(* Logix 5000 project; controller CarbonScout_MK6 vendor 1 type 14 code 154 rev 32.11; software revision 32.00; part 13 of 17 *)
(* tags used below, declared in another part *)
   Data_TLSaver : BOOL;
   DN_Cal : BOOL;   // Calculation Done Bit to proceed next step
   Index : DINT;
   LocalSampleTank : DINT;
   ONS : BOOL[32];
   TimeCompare : TimerCompare;
   AI_LIT_01 : P_AIn;   // Carbon Scout Laser Level Transmitter
   AI_LIT_02 : P_AIn;   // Carbon Scout Cone Level Transmitter
   CS_CarbonSP : REAL;
   CS_DINTParams : DINT[100];
   CS_REALParams : REAL[80];   // CS REAL Parameters
   CS_Result : CS_Results;   // Sample Result Live Async
   CS_Results : CS_Results[20];   // Results Just for DataStore
   CS_ResultStore : CS_Results[20,20];   // Sample Result Historical
   CS_Seq : GEK_Sequence;
   CS_Seq_ControlStop : BOOL;
   CS_Tank : CS_TankParams[20];
   CS_Timer : TIMER[80];
   Data_constant1 : BOOL;
   Data_Saved : BOOL;
   Data_Saver : BOOL;
   Data_Trigger : BOOL;
   Data_Triggered : BOOL;
   Delete2_Trigger : BOOL;
   Delete_Trigger : BOOL;
   Email_Trigger : BOOL;
   Email_Trigger2 : BOOL;
   LeakCheck : BOOL;
   N51 : DINT[5];   // From Client
   Oneshot : DINT;
   Oneshot2 : DINT;
   Oneshot3 : DINT;
   Simulation : DINT;
   TankNum : DINT;
   TankPointer : DINT;
   TimeAndDate : DINT[7];
   Valve_XV_19 : P_ValveSO;   // Laser window
(* SeqProgram, continued *)

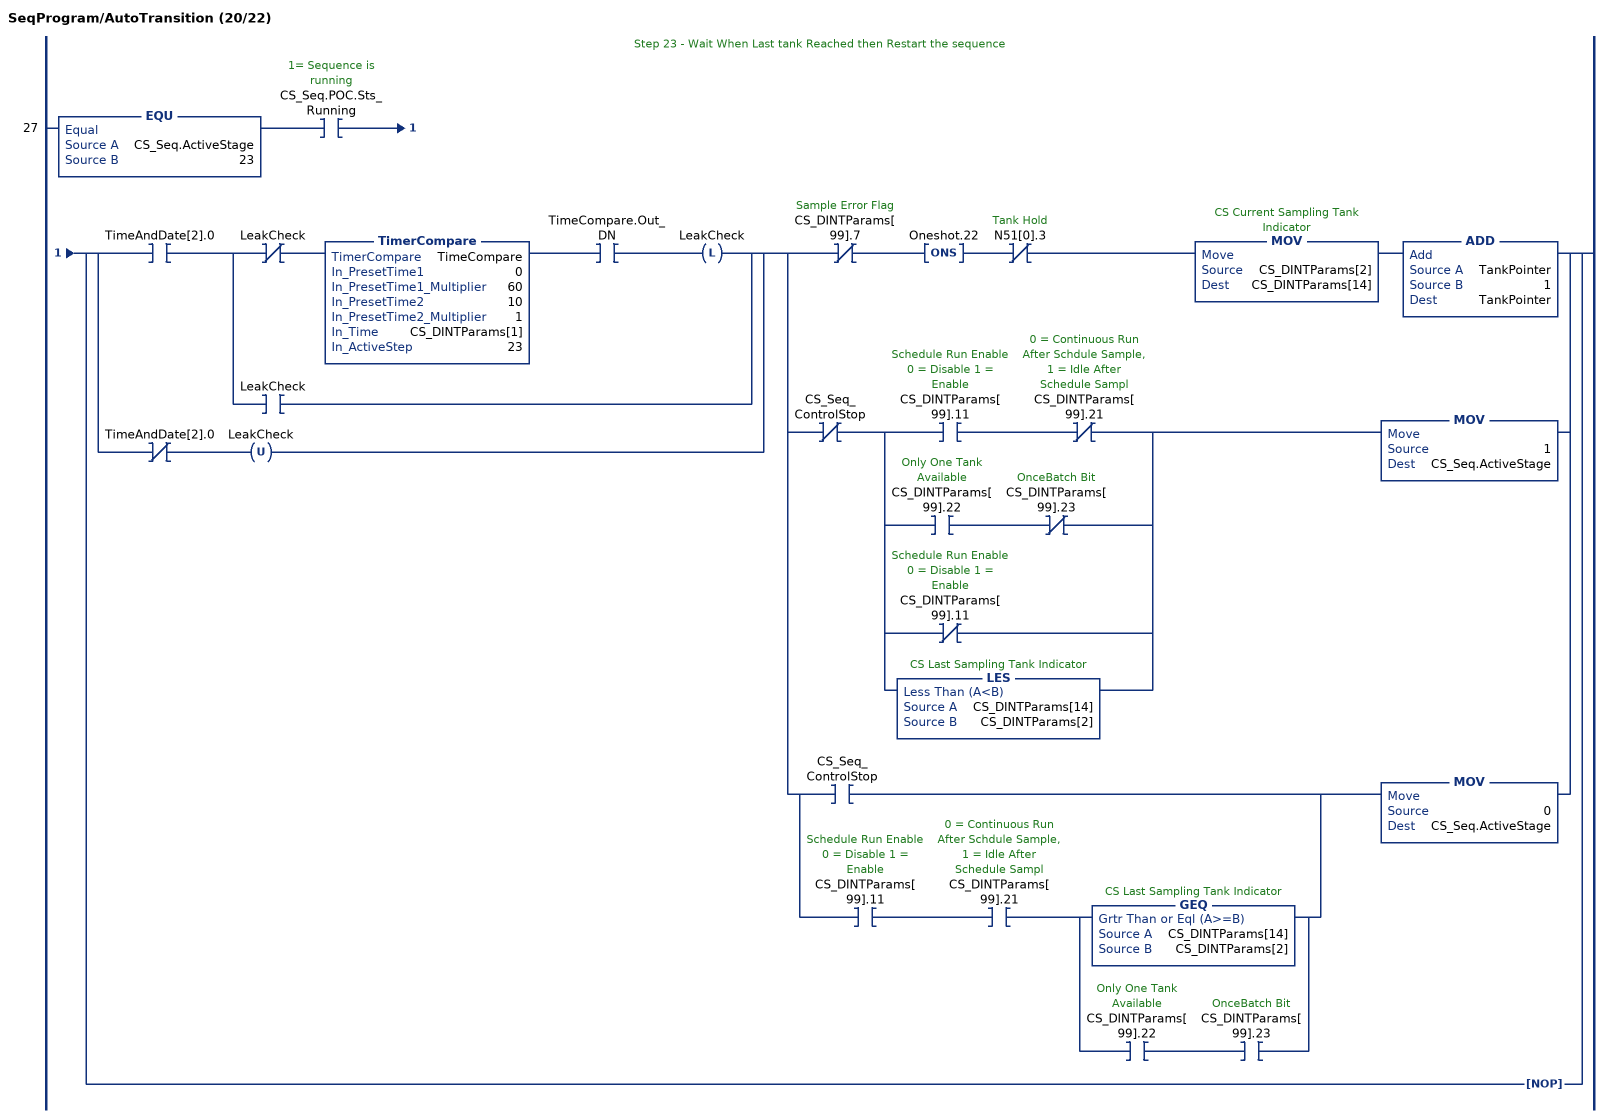
   [picture p263: SeqProgram/AutoTransition rungs 27-27]
   // Step 23 - Wait When Last tank Reached then Restart the sequence
   27: EQU(CS_Seq.ActiveStage,23)XIC(CS_Seq.POC.Sts_Running)[[XIC(TimeAndDate[2].0) [XIO(LeakCheck) TimerCompare(TimeCompare,0,60,10,1,CS_DINTParams[1],23) XIC(TimeCompare.Out_DN) OTL(LeakCheck) ,XIC(LeakCheck) ] ,XIO(TimeAndDate[2].0) OTU(LeakCheck) ] [XIO(CS_DINTParams[99].7) ONS(Oneshot.22) XIO(N51[0].3) MOV(CS_DINTParams[2],CS_DINTParams[14]) ADD(TankPointer,1,TankPointer) ,[XIO(CS_Seq_ControlStop) [XIC(CS_DINTParams[99].11) XIO(CS_DINTParams[99].21) ,[XIC(CS_DINTParams[99].22) XIO(CS_DINTParams[99].23) ,XIO(CS_DINTParams[99].11) ,LES(CS_DINTParams[14],CS_DINTParams[2]) ] ] MOV(1,CS_Seq.ActiveStage) ,[XIC(CS_Seq_ControlStop) ,XIC(CS_DINTParams[99].11) XIC(CS_DINTParams[99].21) [GEQ(CS_DINTParams[14],CS_DINTParams[2]) ,XIC(CS_DINTParams[99].22) XIC(CS_DINTParams[99].23) ] ] MOV(0,CS_Seq.ActiveStage) ] ] ,NOP() ];
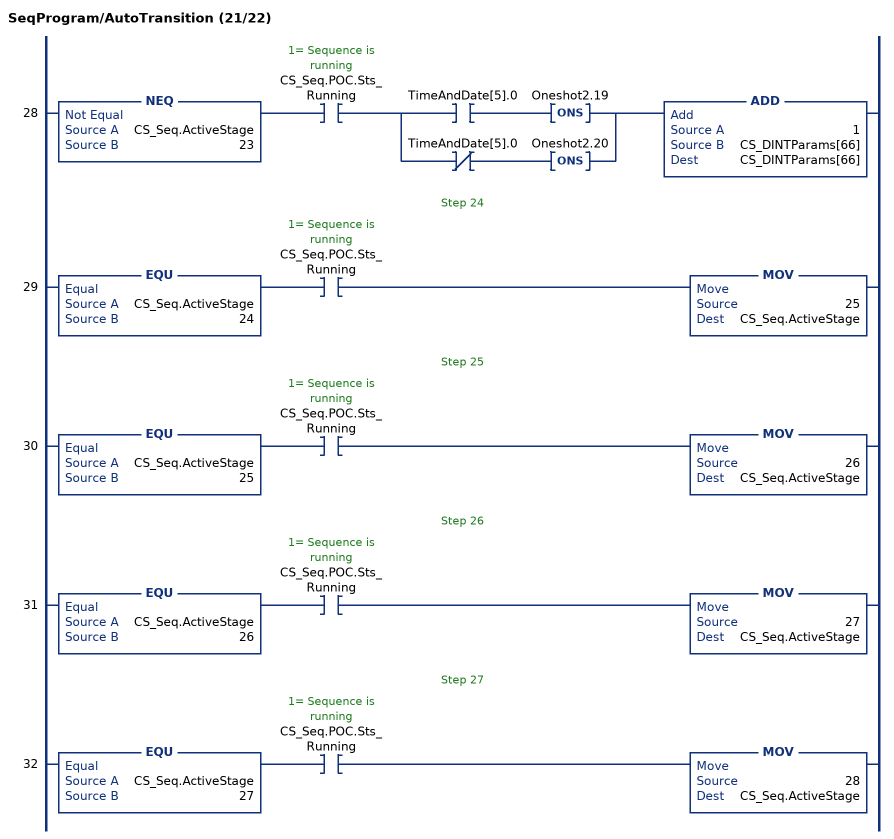
   28: NEQ(CS_Seq.ActiveStage,23)XIC(CS_Seq.POC.Sts_Running)[XIC(TimeAndDate[5].0) ONS(Oneshot2.19) ,XIO(TimeAndDate[5].0) ONS(Oneshot2.20) ]ADD(1,CS_DINTParams[66],CS_DINTParams[66]);
   // Step 24
   29: EQU(CS_Seq.ActiveStage,24)XIC(CS_Seq.POC.Sts_Running)MOV(25,CS_Seq.ActiveStage);
   // Step 25
   30: EQU(CS_Seq.ActiveStage,25)XIC(CS_Seq.POC.Sts_Running)MOV(26,CS_Seq.ActiveStage);
   // Step 26
   31: EQU(CS_Seq.ActiveStage,26)XIC(CS_Seq.POC.Sts_Running)MOV(27,CS_Seq.ActiveStage);
   // Step 27
   32: EQU(CS_Seq.ActiveStage,27)XIC(CS_Seq.POC.Sts_Running)MOV(28,CS_Seq.ActiveStage);
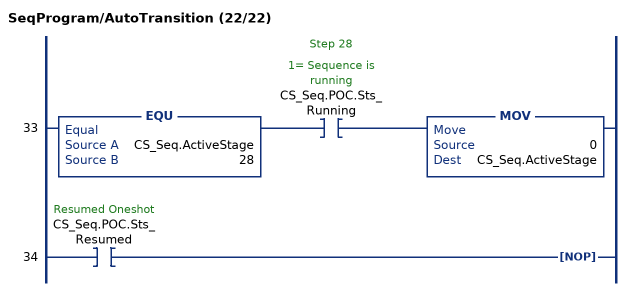
   // Step 28
   33: EQU(CS_Seq.ActiveStage,28)XIC(CS_Seq.POC.Sts_Running)MOV(0,CS_Seq.ActiveStage);
   34: XIC(CS_Seq.POC.Sts_Resumed)NOP();
END_ROUTINE

ROUTINE CarbonCals   (* ladder *)
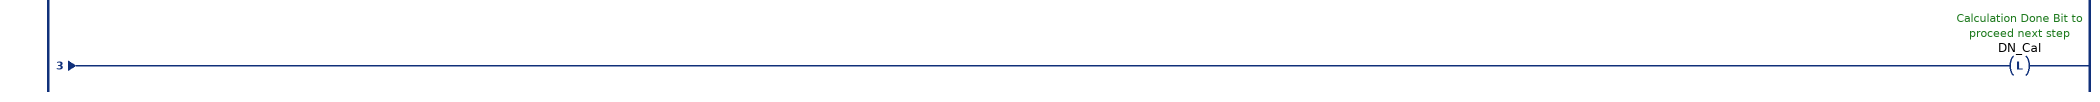
   // Calculating carbon volume
   0: EQU(CS_Seq.ActiveStage,14)XIO(CS_Tank[LocalSampleTank].LeachOnly)XIC(CS_Seq.POC.Sts_Running)[XIC(TimeCompare.Out_DN) [XIO(CS_DINTParams[93].20) [XIC(CS_DINTParams[93].8) ,XIC(CS_DINTParams[93].9) ] ,XIO(CS_DINTParams[99].15) ] ,XIC(CS_Timer[71].EN) ]TON(CS_Timer[71],?,?)XIC(CS_Timer[71].DN)ONS(Oneshot.23)[CPT(CS_REALParams[15],CS_REALParams[0]-CS_REALParams[1]) [CMP(CS_REALParams[15]<=0) CLR(CS_Result.Carbon_VOL_ml) ,CMP(CS_REALParams[15]>0) [CMP(CS_REALParams[15]<=CS_REALParams[14]) CPT(CS_Result.Carbon_VOL_ml,CS_REALParams[15]*(CS_REALParams[5]*CS_REALParams[5]/4)*3.1415927/1000) ,CMP(CS_REALParams[15]>CS_REALParams[14]) [CPT(CS_REALParams[17],CS_REALParams[14]*(CS_REALParams[5]*CS_REALParams[5]/4)*3.1415927) ,CPT(CS_REALParams[19],CS_REALParams[13]-CS_REALParams[14]) ,CPT(CS_REALParams[21],CS_REALParams[19]/(CS_REALParams[12]-CS_REALParams[5])) ,CPT(CS_REALParams[16],CS_REALParams[5]*CS_REALParams[21]) ,CPT(CS_REALParams[20],CS_REALParams[16]+(CS_REALParams[15]-CS_REALParams[14])) ,CPT(CS_REALParams[18],CS_REALParams[20]/CS_REALParams[21]) ] CPT(CS_Result.Carbon_VOL_ml,(CS_REALParams[17]+((CS_REALParams[18]*CS_REALParams[18]*3.1415927/4*CS_REALParams[20]-(CS_REALParams[5]*CS_REALParams[5]*3.1415927/4*CS_REALParams[16]))/3))/1000) ] ] ,DIV(CS_Result.Carbon_VOL_ml,CS_REALParams[11],CS_REALParams[51]) MOV(CS_REALParams[51],CS_Result.Carbon_mLperL) MUL(CS_Result.Carbon_VOL_ml,CS_REALParams[6],CS_Result.Carbon_MASS) ,MOV(LocalSampleTank,CS_Result.Sample_Tank) MOV(CS_REALParams[15],CS_Result.Carbon_Height) DIV(CS_Result.Carbon_MASS,CS_REALParams[11],CS_Result.Carbon_DIST) CPT(CS_Tank[LocalSampleTank].TotalCarbonMass,CS_Result.Carbon_DIST*CS_Tank[LocalSampleTank].Volume) CPT(CS_Tank[LocalSampleTank].GoldMass,CS_Tank[LocalSampleTank].TotalCarbonMass*CS_Result.Au) CPT(CS_Result.DisplacedCarbonVol,CS_REALParams[51]*(CS_Result.Sample_FlowRate*CS_Tank[LocalSampleTank].Sample_Time*0.4)) CPT(CS_Result.DisplacedCarbonMass,CS_Result.Sample_FlowRate*CS_Tank[LocalSampleTank].Sample_Time*0.4*CS_Result.Carbon_DIST) ,MOV(TimeAndDate[0],CS_Result.Year) MOV(TimeAndDate[1],CS_Result.Month) MOV(TimeAndDate[2],CS_Result.Day) MOV(TimeAndDate[3],CS_Result.Hour) MOV(TimeAndDate[4],CS_Result.Min) ,MOV(0,Index) FOR(DataShift,Index,0,18,1) CPS(CS_Result,CS_ResultStore[LocalSampleTank,0],1) ]OTL(DN_Cal);
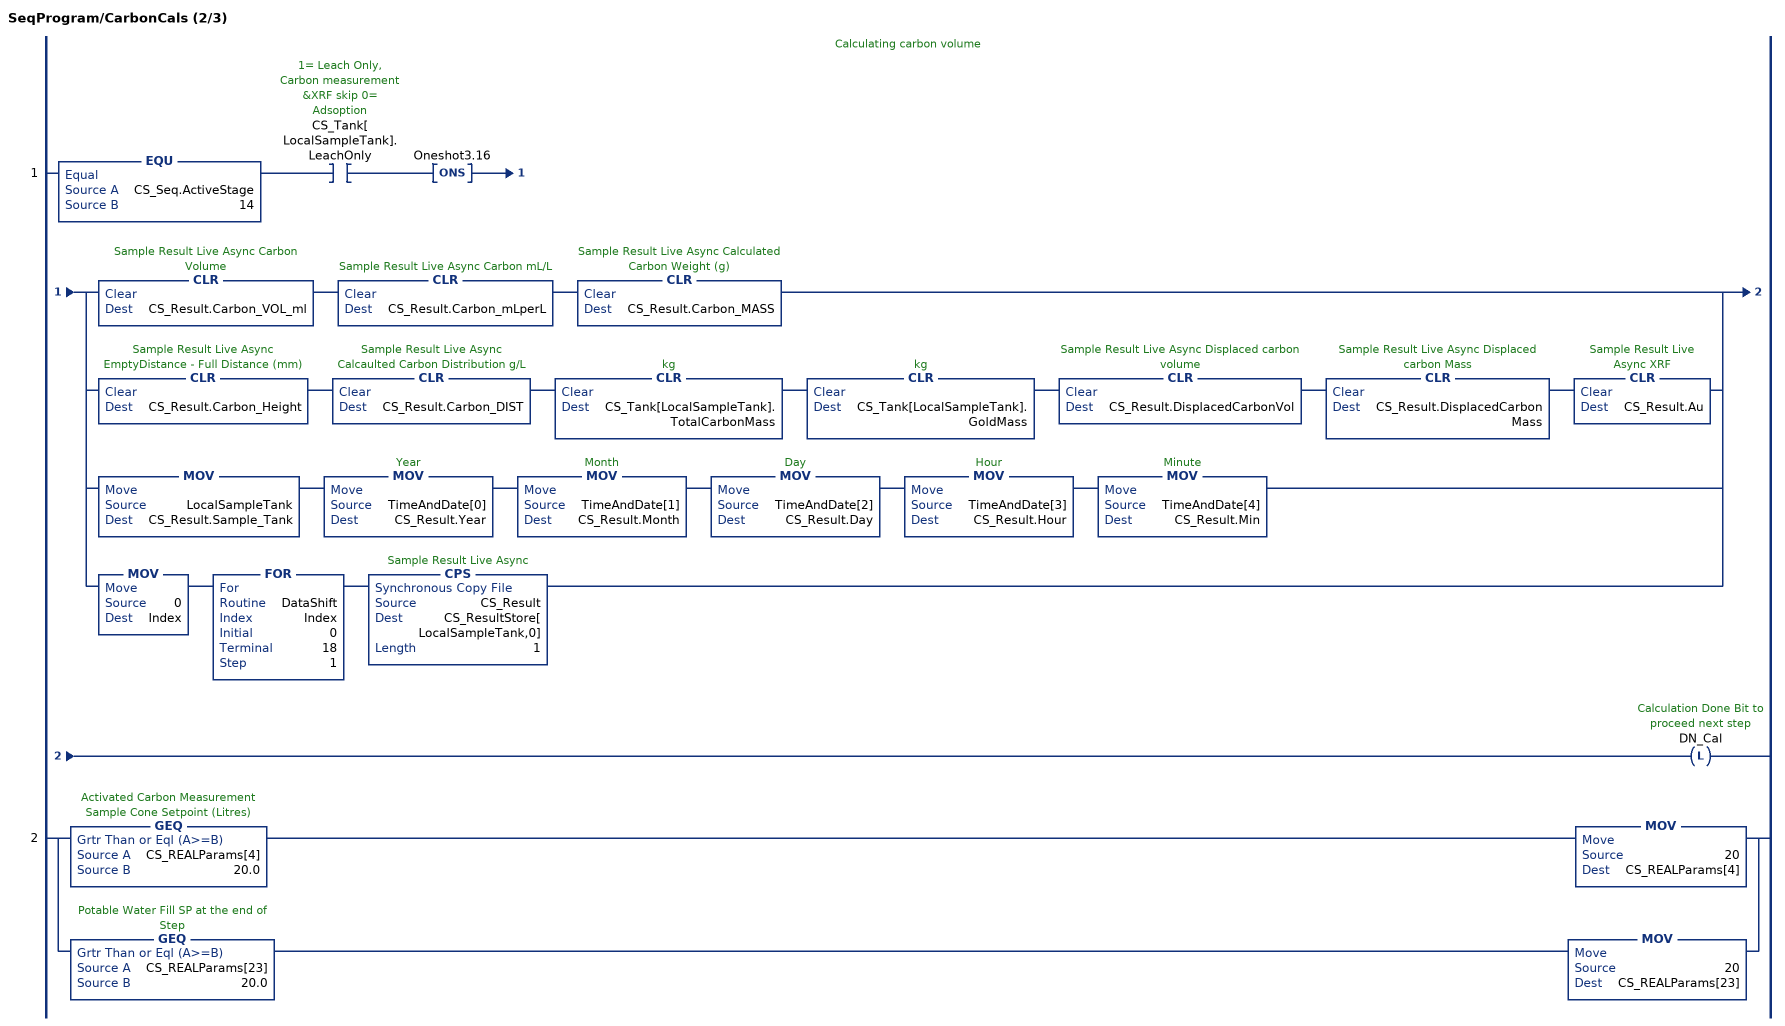
   // Calculating carbon volume
   1: EQU(CS_Seq.ActiveStage,14)XIC(CS_Tank[LocalSampleTank].LeachOnly)ONS(Oneshot3.16)[CLR(CS_Result.Carbon_VOL_ml) CLR(CS_Result.Carbon_mLperL) CLR(CS_Result.Carbon_MASS) ,CLR(CS_Result.Carbon_Height) CLR(CS_Result.Carbon_DIST) CLR(CS_Tank[LocalSampleTank].TotalCarbonMass) CLR(CS_Tank[LocalSampleTank].GoldMass) CLR(CS_Result.DisplacedCarbonVol) CLR(CS_Result.DisplacedCarbonMass) CLR(CS_Result.Au) ,MOV(LocalSampleTank,CS_Result.Sample_Tank) MOV(TimeAndDate[0],CS_Result.Year) MOV(TimeAndDate[1],CS_Result.Month) MOV(TimeAndDate[2],CS_Result.Day) MOV(TimeAndDate[3],CS_Result.Hour) MOV(TimeAndDate[4],CS_Result.Min) ,MOV(0,Index) FOR(DataShift,Index,0,18,1) CPS(CS_Result,CS_ResultStore[LocalSampleTank,0],1) ]OTL(DN_Cal);
   2: [GEQ(CS_REALParams[4],20.0) MOV(20,CS_REALParams[4]) ,GEQ(CS_REALParams[23],20.0) MOV(20,CS_REALParams[23]) ];
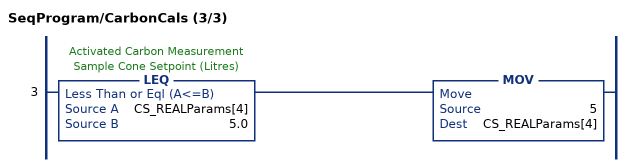
   3: LEQ(CS_REALParams[4],5.0)MOV(5,CS_REALParams[4]);
END_ROUTINE

ROUTINE Commissioning_ParamCalculation   (* ladder *)
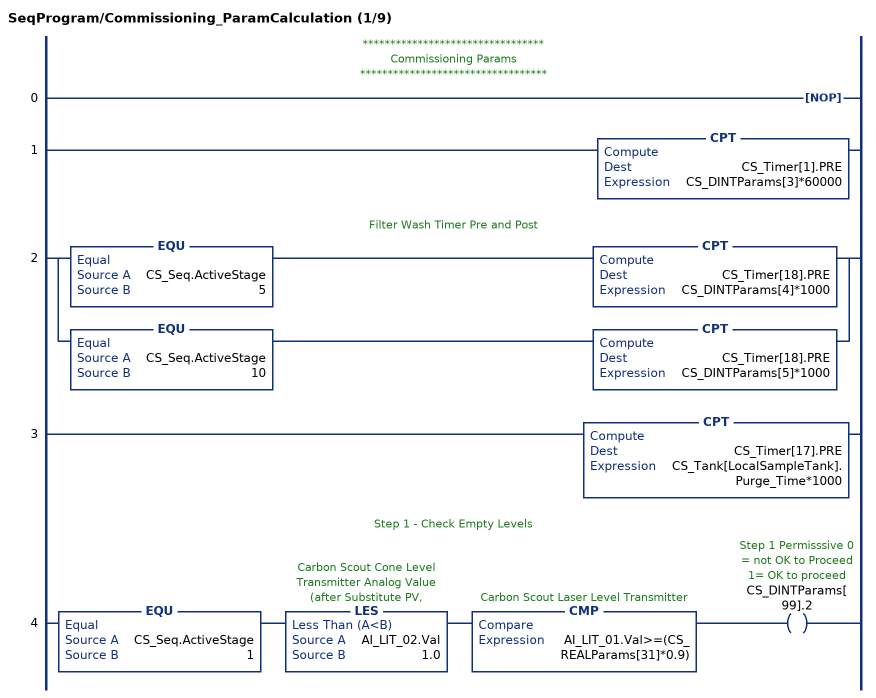
   // *********************************
   // Commissioning Params
   // **********************************
   0: NOP();
   1: CPT(CS_Timer[1].PRE,CS_DINTParams[3]*60000);
   // Filter Wash Timer Pre and Post
   2: [EQU(CS_Seq.ActiveStage,5) CPT(CS_Timer[18].PRE,CS_DINTParams[4]*1000) ,EQU(CS_Seq.ActiveStage,10) CPT(CS_Timer[18].PRE,CS_DINTParams[5]*1000) ];
   3: CPT(CS_Timer[17].PRE,CS_Tank[LocalSampleTank].Purge_Time*1000);
   // Step 1 - Check Empty Levels
   4: EQU(CS_Seq.ActiveStage,1)LES(AI_LIT_02.Val,1.0)CMP(AI_LIT_01.Val>=(CS_REALParams[31]*0.9))OTE(CS_DINTParams[99].2);
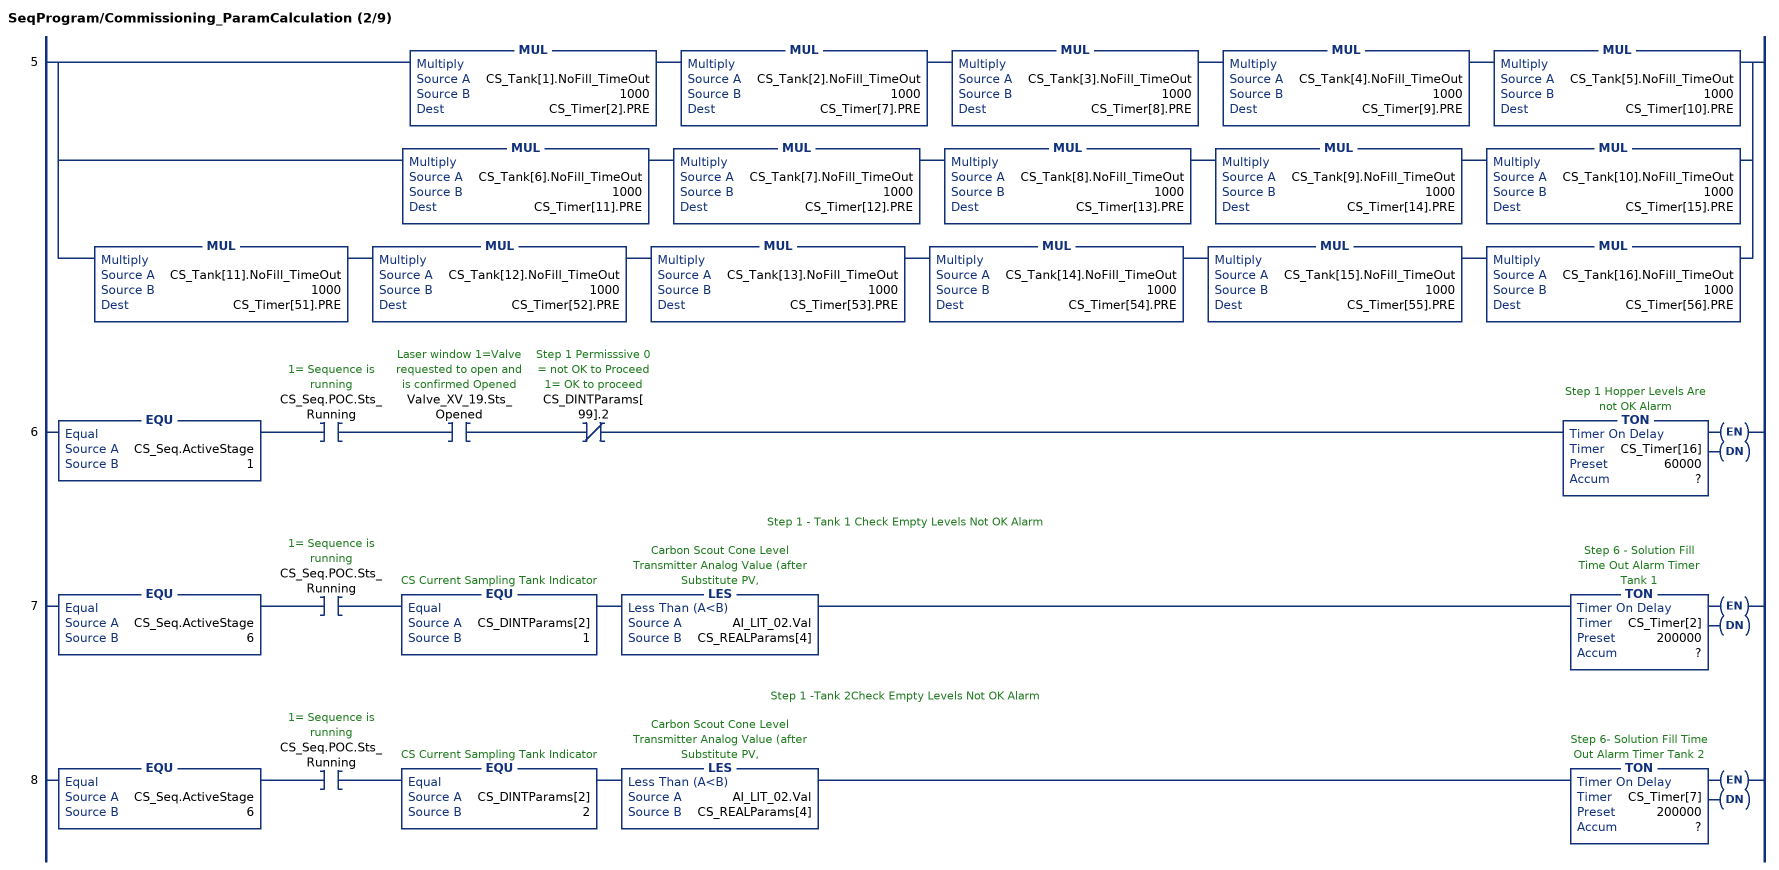
   5: [MUL(CS_Tank[1].NoFill_TimeOut,1000,CS_Timer[2].PRE) MUL(CS_Tank[2].NoFill_TimeOut,1000,CS_Timer[7].PRE) MUL(CS_Tank[3].NoFill_TimeOut,1000,CS_Timer[8].PRE) MUL(CS_Tank[4].NoFill_TimeOut,1000,CS_Timer[9].PRE) MUL(CS_Tank[5].NoFill_TimeOut,1000,CS_Timer[10].PRE) ,MUL(CS_Tank[6].NoFill_TimeOut,1000,CS_Timer[11].PRE) MUL(CS_Tank[7].NoFill_TimeOut,1000,CS_Timer[12].PRE) MUL(CS_Tank[8].NoFill_TimeOut,1000,CS_Timer[13].PRE) MUL(CS_Tank[9].NoFill_TimeOut,1000,CS_Timer[14].PRE) MUL(CS_Tank[10].NoFill_TimeOut,1000,CS_Timer[15].PRE) ,MUL(CS_Tank[11].NoFill_TimeOut,1000,CS_Timer[51].PRE) MUL(CS_Tank[12].NoFill_TimeOut,1000,CS_Timer[52].PRE) MUL(CS_Tank[13].NoFill_TimeOut,1000,CS_Timer[53].PRE) MUL(CS_Tank[14].NoFill_TimeOut,1000,CS_Timer[54].PRE) MUL(CS_Tank[15].NoFill_TimeOut,1000,CS_Timer[55].PRE) MUL(CS_Tank[16].NoFill_TimeOut,1000,CS_Timer[56].PRE) ];
   6: EQU(CS_Seq.ActiveStage,1)XIC(CS_Seq.POC.Sts_Running)XIC(Valve_XV_19.Sts_Opened)XIO(CS_DINTParams[99].2)TON(CS_Timer[16],?,?);
   // Step 1 - Tank 1 Check Empty Levels Not OK Alarm
   7: EQU(CS_Seq.ActiveStage,6)XIC(CS_Seq.POC.Sts_Running)EQU(CS_DINTParams[2],1)LES(AI_LIT_02.Val,CS_REALParams[4])TON(CS_Timer[2],?,?);
   // Step 1 -Tank 2Check Empty Levels Not OK Alarm
   8: EQU(CS_Seq.ActiveStage,6)XIC(CS_Seq.POC.Sts_Running)EQU(CS_DINTParams[2],2)LES(AI_LIT_02.Val,CS_REALParams[4])TON(CS_Timer[7],?,?);
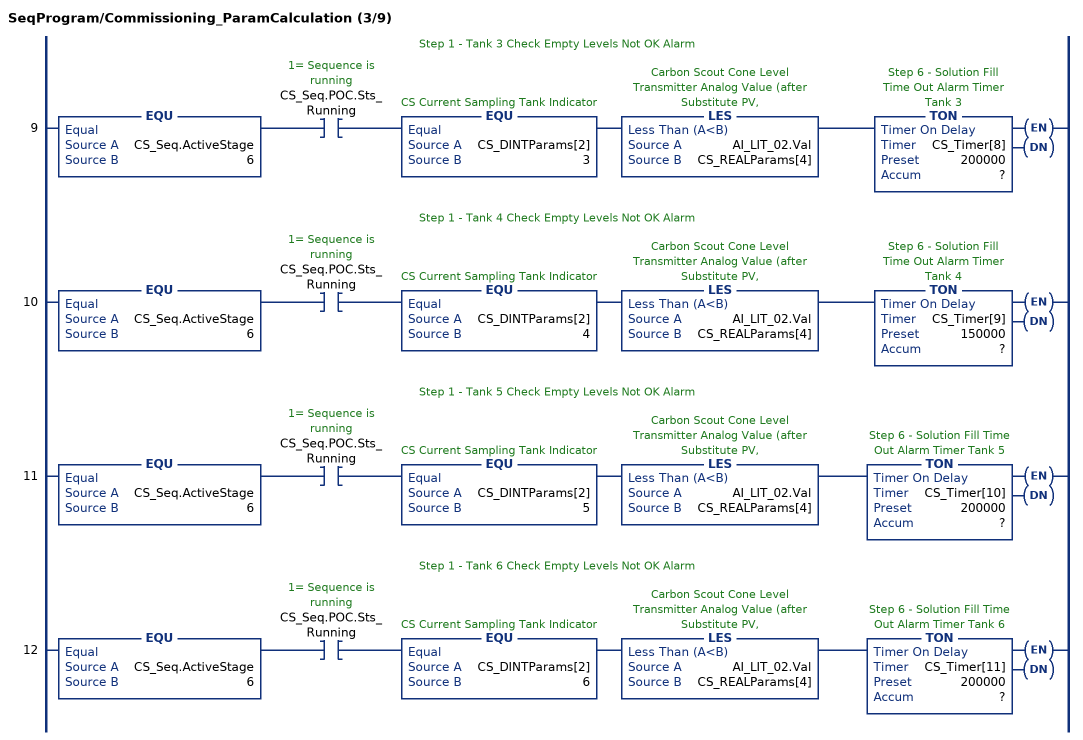
   // Step 1 - Tank 3 Check Empty Levels Not OK Alarm
   9: EQU(CS_Seq.ActiveStage,6)XIC(CS_Seq.POC.Sts_Running)EQU(CS_DINTParams[2],3)LES(AI_LIT_02.Val,CS_REALParams[4])TON(CS_Timer[8],?,?);
   // Step 1 - Tank 4 Check Empty Levels Not OK Alarm
   10: EQU(CS_Seq.ActiveStage,6)XIC(CS_Seq.POC.Sts_Running)EQU(CS_DINTParams[2],4)LES(AI_LIT_02.Val,CS_REALParams[4])TON(CS_Timer[9],?,?);
   // Step 1 - Tank 5 Check Empty Levels Not OK Alarm
   11: EQU(CS_Seq.ActiveStage,6)XIC(CS_Seq.POC.Sts_Running)EQU(CS_DINTParams[2],5)LES(AI_LIT_02.Val,CS_REALParams[4])TON(CS_Timer[10],?,?);
   // Step 1 - Tank 6 Check Empty Levels Not OK Alarm
   12: EQU(CS_Seq.ActiveStage,6)XIC(CS_Seq.POC.Sts_Running)EQU(CS_DINTParams[2],6)LES(AI_LIT_02.Val,CS_REALParams[4])TON(CS_Timer[11],?,?);
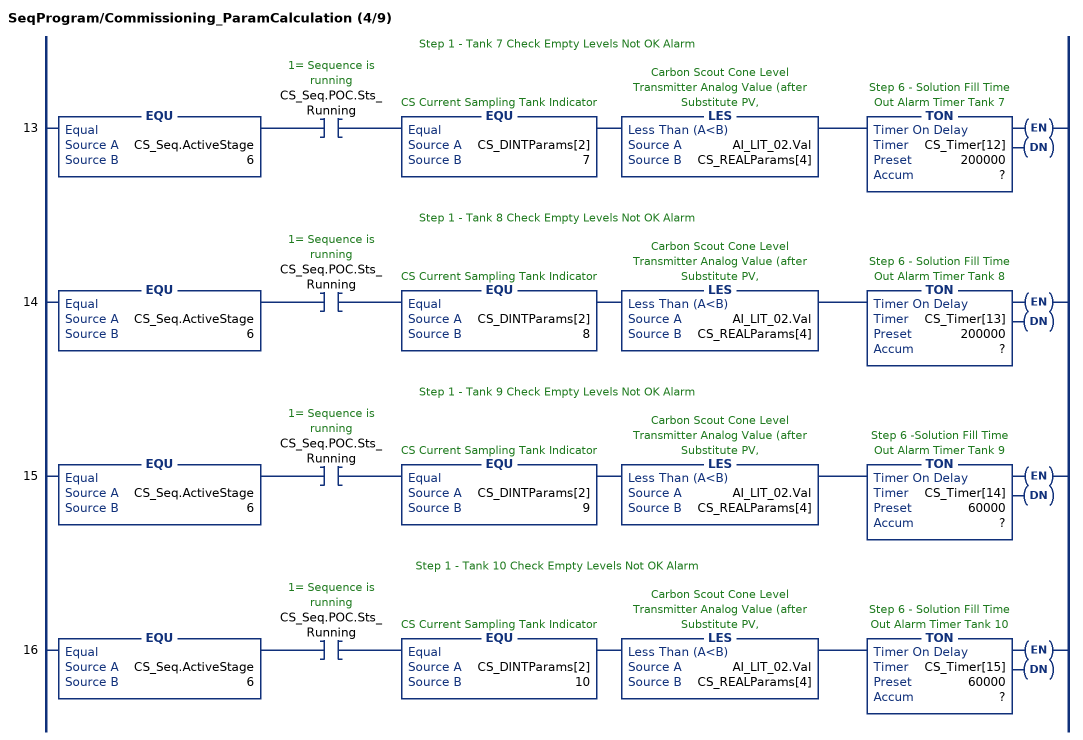
   // Step 1 - Tank 7 Check Empty Levels Not OK Alarm
   13: EQU(CS_Seq.ActiveStage,6)XIC(CS_Seq.POC.Sts_Running)EQU(CS_DINTParams[2],7)LES(AI_LIT_02.Val,CS_REALParams[4])TON(CS_Timer[12],?,?);
   // Step 1 - Tank 8 Check Empty Levels Not OK Alarm
   14: EQU(CS_Seq.ActiveStage,6)XIC(CS_Seq.POC.Sts_Running)EQU(CS_DINTParams[2],8)LES(AI_LIT_02.Val,CS_REALParams[4])TON(CS_Timer[13],?,?);
   // Step 1 - Tank 9 Check Empty Levels Not OK Alarm
   15: EQU(CS_Seq.ActiveStage,6)XIC(CS_Seq.POC.Sts_Running)EQU(CS_DINTParams[2],9)LES(AI_LIT_02.Val,CS_REALParams[4])TON(CS_Timer[14],?,?);
   // Step 1 - Tank 10 Check Empty Levels Not OK Alarm
   16: EQU(CS_Seq.ActiveStage,6)XIC(CS_Seq.POC.Sts_Running)EQU(CS_DINTParams[2],10)LES(AI_LIT_02.Val,CS_REALParams[4])TON(CS_Timer[15],?,?);
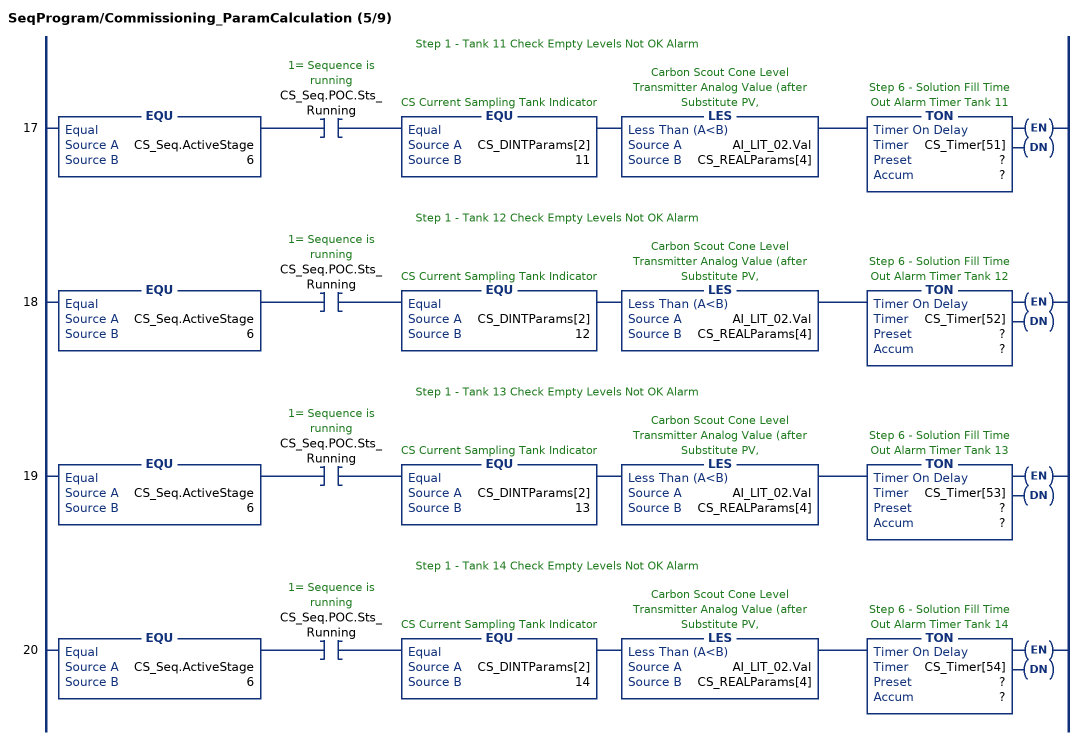
   // Step 1 - Tank 11 Check Empty Levels Not OK Alarm
   17: EQU(CS_Seq.ActiveStage,6)XIC(CS_Seq.POC.Sts_Running)EQU(CS_DINTParams[2],11)LES(AI_LIT_02.Val,CS_REALParams[4])TON(CS_Timer[51],?,?);
   // Step 1 - Tank 12 Check Empty Levels Not OK Alarm
   18: EQU(CS_Seq.ActiveStage,6)XIC(CS_Seq.POC.Sts_Running)EQU(CS_DINTParams[2],12)LES(AI_LIT_02.Val,CS_REALParams[4])TON(CS_Timer[52],?,?);
   // Step 1 - Tank 13 Check Empty Levels Not OK Alarm
   19: EQU(CS_Seq.ActiveStage,6)XIC(CS_Seq.POC.Sts_Running)EQU(CS_DINTParams[2],13)LES(AI_LIT_02.Val,CS_REALParams[4])TON(CS_Timer[53],?,?);
   // Step 1 - Tank 14 Check Empty Levels Not OK Alarm
   20: EQU(CS_Seq.ActiveStage,6)XIC(CS_Seq.POC.Sts_Running)EQU(CS_DINTParams[2],14)LES(AI_LIT_02.Val,CS_REALParams[4])TON(CS_Timer[54],?,?);
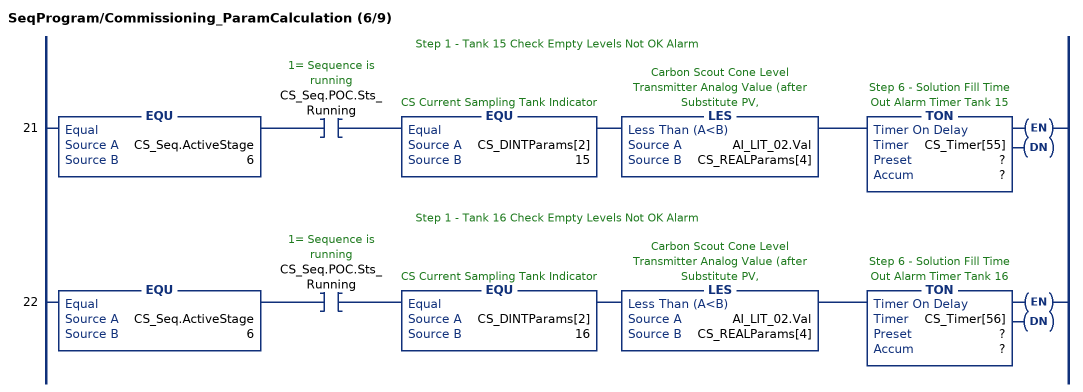
   // Step 1 - Tank 15 Check Empty Levels Not OK Alarm
   21: EQU(CS_Seq.ActiveStage,6)XIC(CS_Seq.POC.Sts_Running)EQU(CS_DINTParams[2],15)LES(AI_LIT_02.Val,CS_REALParams[4])TON(CS_Timer[55],?,?);
   // Step 1 - Tank 16 Check Empty Levels Not OK Alarm
   22: EQU(CS_Seq.ActiveStage,6)XIC(CS_Seq.POC.Sts_Running)EQU(CS_DINTParams[2],16)LES(AI_LIT_02.Val,CS_REALParams[4])TON(CS_Timer[56],?,?);
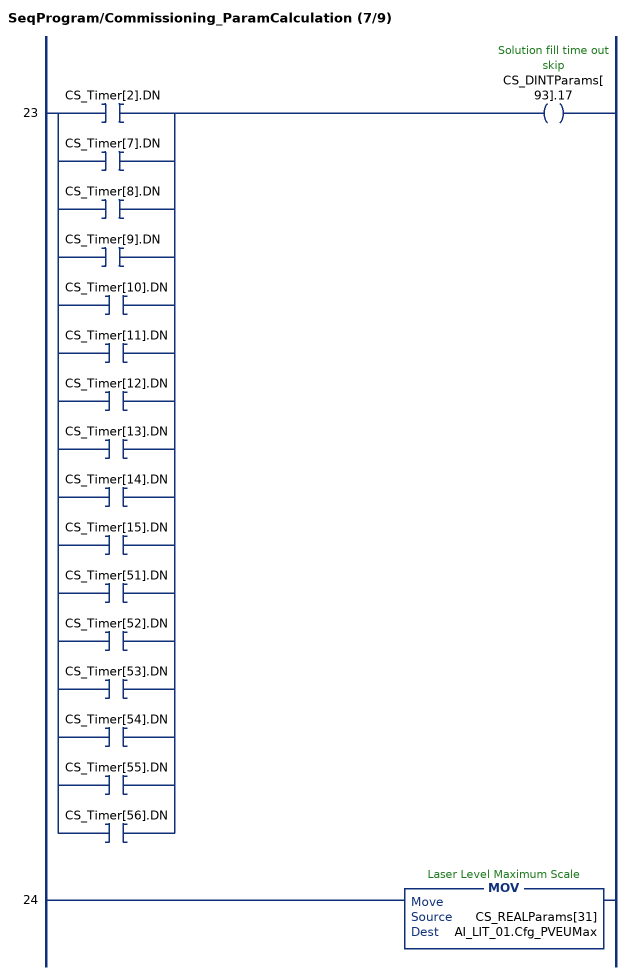
   23: [XIC(CS_Timer[2].DN) ,XIC(CS_Timer[7].DN) ,XIC(CS_Timer[8].DN) ,XIC(CS_Timer[9].DN) ,XIC(CS_Timer[10].DN) ,XIC(CS_Timer[11].DN) ,[XIC(CS_Timer[12].DN) ,XIC(CS_Timer[13].DN) ,XIC(CS_Timer[14].DN) ,XIC(CS_Timer[15].DN) ,XIC(CS_Timer[51].DN) ,XIC(CS_Timer[52].DN) ,XIC(CS_Timer[53].DN) ,XIC(CS_Timer[54].DN) ,XIC(CS_Timer[55].DN) ,XIC(CS_Timer[56].DN) ] ]OTE(CS_DINTParams[93].17);
   24: MOV(CS_REALParams[31],AI_LIT_01.Cfg_PVEUMax);
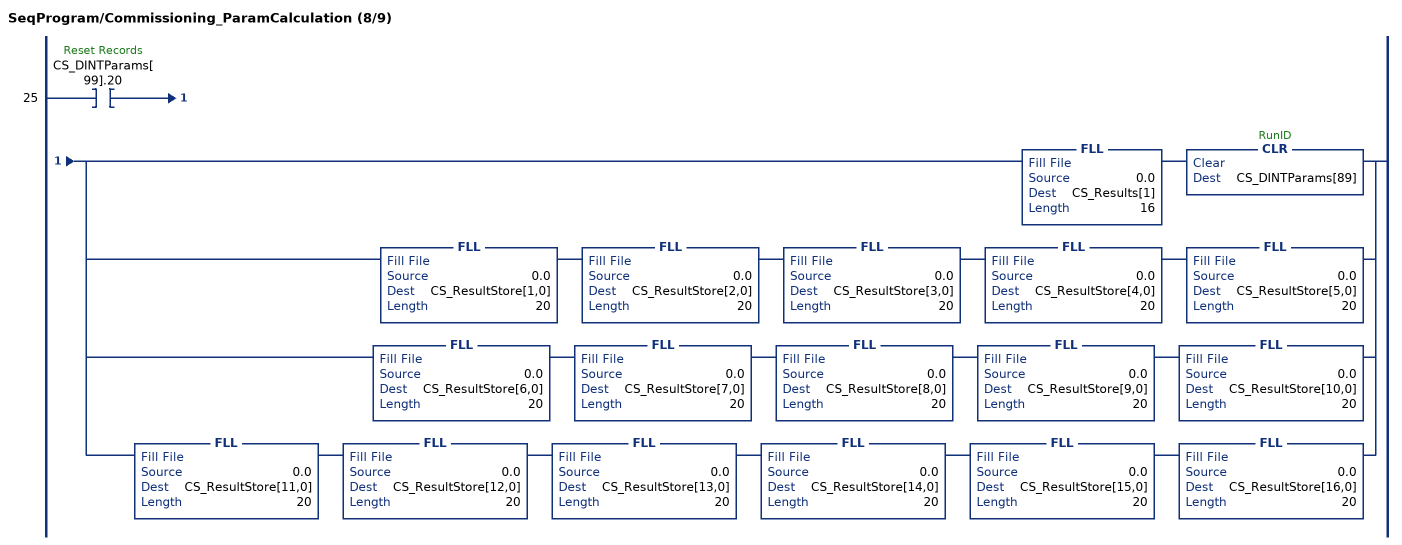
   25: XIC(CS_DINTParams[99].20)[FLL(0.0,CS_Results[1],16) CLR(CS_DINTParams[89]) ,FLL(0.0,CS_ResultStore[1,0],20) FLL(0.0,CS_ResultStore[2,0],20) FLL(0.0,CS_ResultStore[3,0],20) FLL(0.0,CS_ResultStore[4,0],20) FLL(0.0,CS_ResultStore[5,0],20) ,FLL(0.0,CS_ResultStore[6,0],20) FLL(0.0,CS_ResultStore[7,0],20) FLL(0.0,CS_ResultStore[8,0],20) FLL(0.0,CS_ResultStore[9,0],20) FLL(0.0,CS_ResultStore[10,0],20) ,FLL(0.0,CS_ResultStore[11,0],20) FLL(0.0,CS_ResultStore[12,0],20) FLL(0.0,CS_ResultStore[13,0],20) FLL(0.0,CS_ResultStore[14,0],20) FLL(0.0,CS_ResultStore[15,0],20) FLL(0.0,CS_ResultStore[16,0],20) ];
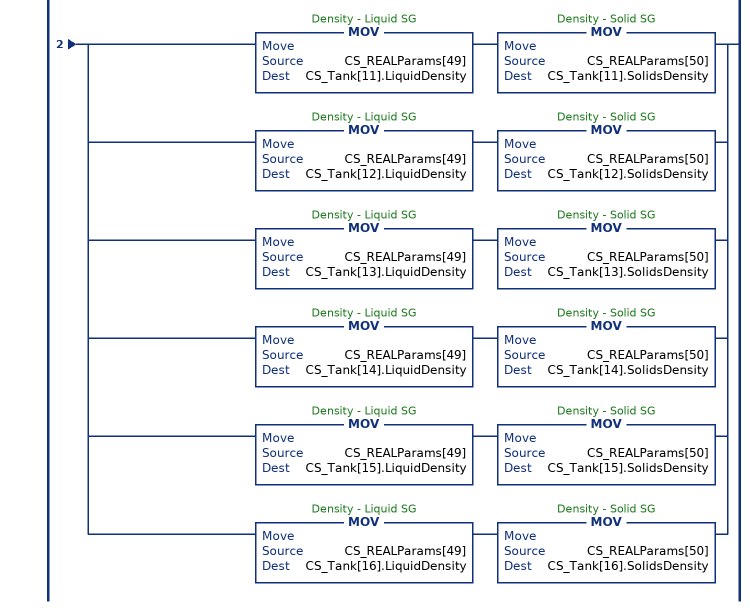
   26: XIC(CS_DINTParams[99].17)[MOV(CS_REALParams[49],CS_Tank[1].LiquidDensity) MOV(CS_REALParams[50],CS_Tank[1].SolidsDensity) ,MOV(CS_REALParams[49],CS_Tank[2].LiquidDensity) MOV(CS_REALParams[50],CS_Tank[2].SolidsDensity) ,MOV(CS_REALParams[49],CS_Tank[3].LiquidDensity) MOV(CS_REALParams[50],CS_Tank[3].SolidsDensity) ,MOV(CS_REALParams[49],CS_Tank[4].LiquidDensity) MOV(CS_REALParams[50],CS_Tank[4].SolidsDensity) ,MOV(CS_REALParams[49],CS_Tank[5].LiquidDensity) MOV(CS_REALParams[50],CS_Tank[5].SolidsDensity) ][MOV(CS_REALParams[49],CS_Tank[6].LiquidDensity) MOV(CS_REALParams[50],CS_Tank[6].SolidsDensity) ,MOV(CS_REALParams[49],CS_Tank[7].LiquidDensity) MOV(CS_REALParams[50],CS_Tank[7].SolidsDensity) ,MOV(CS_REALParams[49],CS_Tank[8].LiquidDensity) MOV(CS_REALParams[50],CS_Tank[8].SolidsDensity) ,MOV(CS_REALParams[49],CS_Tank[9].LiquidDensity) MOV(CS_REALParams[50],CS_Tank[9].SolidsDensity) ,MOV(CS_REALParams[49],CS_Tank[10].LiquidDensity) MOV(CS_REALParams[50],CS_Tank[10].SolidsDensity) ][MOV(CS_REALParams[49],CS_Tank[11].LiquidDensity) MOV(CS_REALParams[50],CS_Tank[11].SolidsDensity) ,MOV(CS_REALParams[49],CS_Tank[12].LiquidDensity) MOV(CS_REALParams[50],CS_Tank[12].SolidsDensity) ,MOV(CS_REALParams[49],CS_Tank[13].LiquidDensity) MOV(CS_REALParams[50],CS_Tank[13].SolidsDensity) ,MOV(CS_REALParams[49],CS_Tank[14].LiquidDensity) MOV(CS_REALParams[50],CS_Tank[14].SolidsDensity) ,MOV(CS_REALParams[49],CS_Tank[15].LiquidDensity) MOV(CS_REALParams[50],CS_Tank[15].SolidsDensity) ,MOV(CS_REALParams[49],CS_Tank[16].LiquidDensity) MOV(CS_REALParams[50],CS_Tank[16].SolidsDensity) ];
END_ROUTINE

ROUTINE DataLogging   (* ladder *)
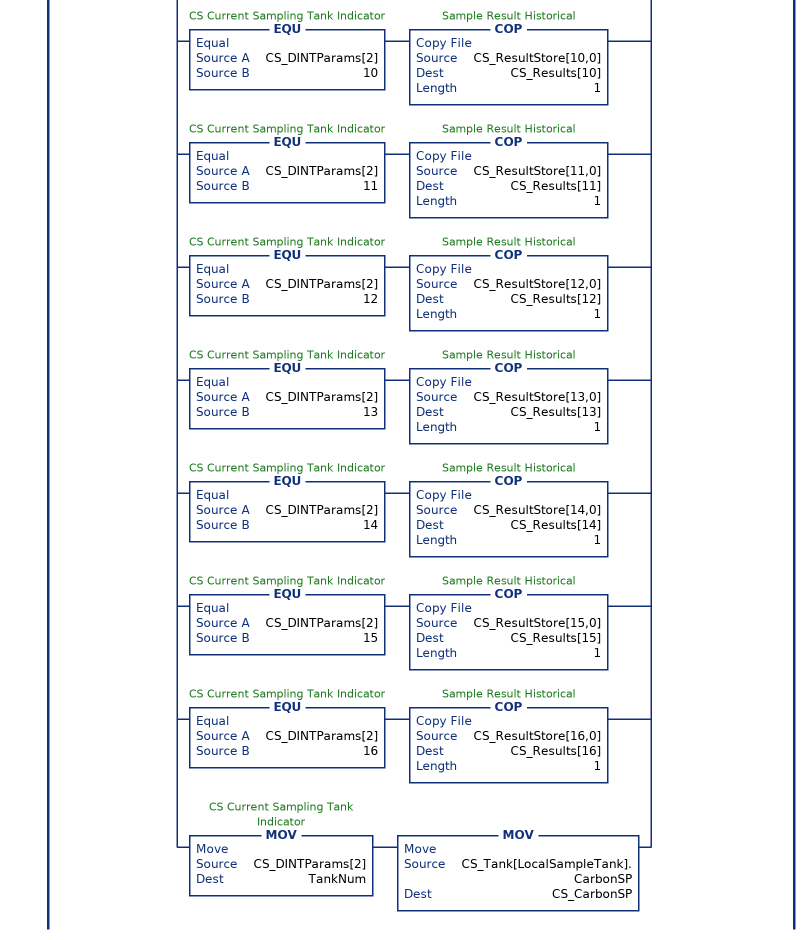
   0: [XIC(CS_Tank[1].LogTrigger) ,XIC(CS_Tank[2].LogTrigger) ,XIC(CS_Tank[3].LogTrigger) ,XIC(CS_Tank[4].LogTrigger) ,XIC(CS_Tank[5].LogTrigger) ,XIC(CS_Tank[6].LogTrigger) ,XIC(CS_Tank[7].LogTrigger) ,XIC(CS_Tank[8].LogTrigger) ,XIC(CS_Tank[9].LogTrigger) ,XIC(CS_Tank[10].LogTrigger) ,XIC(CS_Tank[11].LogTrigger) ,XIC(CS_Tank[12].LogTrigger) ,XIC(CS_Tank[13].LogTrigger) ,XIC(CS_Tank[14].LogTrigger) ,XIC(CS_Tank[15].LogTrigger) ,XIC(CS_Tank[16].LogTrigger) ][[EQU(CS_DINTParams[2],1) COP(CS_ResultStore[1,0],CS_Results[1],1) ,EQU(CS_DINTParams[2],2) COP(CS_ResultStore[2,0],CS_Results[2],1) ,EQU(CS_DINTParams[2],3) COP(CS_ResultStore[3,0],CS_Results[3],1) ,EQU(CS_DINTParams[2],4) COP(CS_ResultStore[4,0],CS_Results[4],1) ,EQU(CS_DINTParams[2],5) COP(CS_ResultStore[5,0],CS_Results[5],1) ,EQU(CS_DINTParams[2],6) COP(CS_ResultStore[6,0],CS_Results[6],1) ,EQU(CS_DINTParams[2],7) COP(CS_ResultStore[7,0],CS_Results[7],1) ,EQU(CS_DINTParams[2],8) COP(CS_ResultStore[8,0],CS_Results[8],1) ,EQU(CS_DINTParams[2],9) COP(CS_ResultStore[9,0],CS_Results[9],1) ,EQU(CS_DINTParams[2],10) COP(CS_ResultStore[10,0],CS_Results[10],1) ,EQU(CS_DINTParams[2],11) COP(CS_ResultStore[11,0],CS_Results[11],1) ,EQU(CS_DINTParams[2],12) COP(CS_ResultStore[12,0],CS_Results[12],1) ,EQU(CS_DINTParams[2],13) COP(CS_ResultStore[13,0],CS_Results[13],1) ,EQU(CS_DINTParams[2],14) COP(CS_ResultStore[14,0],CS_Results[14],1) ,EQU(CS_DINTParams[2],15) COP(CS_ResultStore[15,0],CS_Results[15],1) ,EQU(CS_DINTParams[2],16) COP(CS_ResultStore[16,0],CS_Results[16],1) ] ,MOV(CS_DINTParams[2],TankNum) MOV(CS_Tank[LocalSampleTank].CarbonSP,CS_CarbonSP) ]OTE(Data_Triggered);
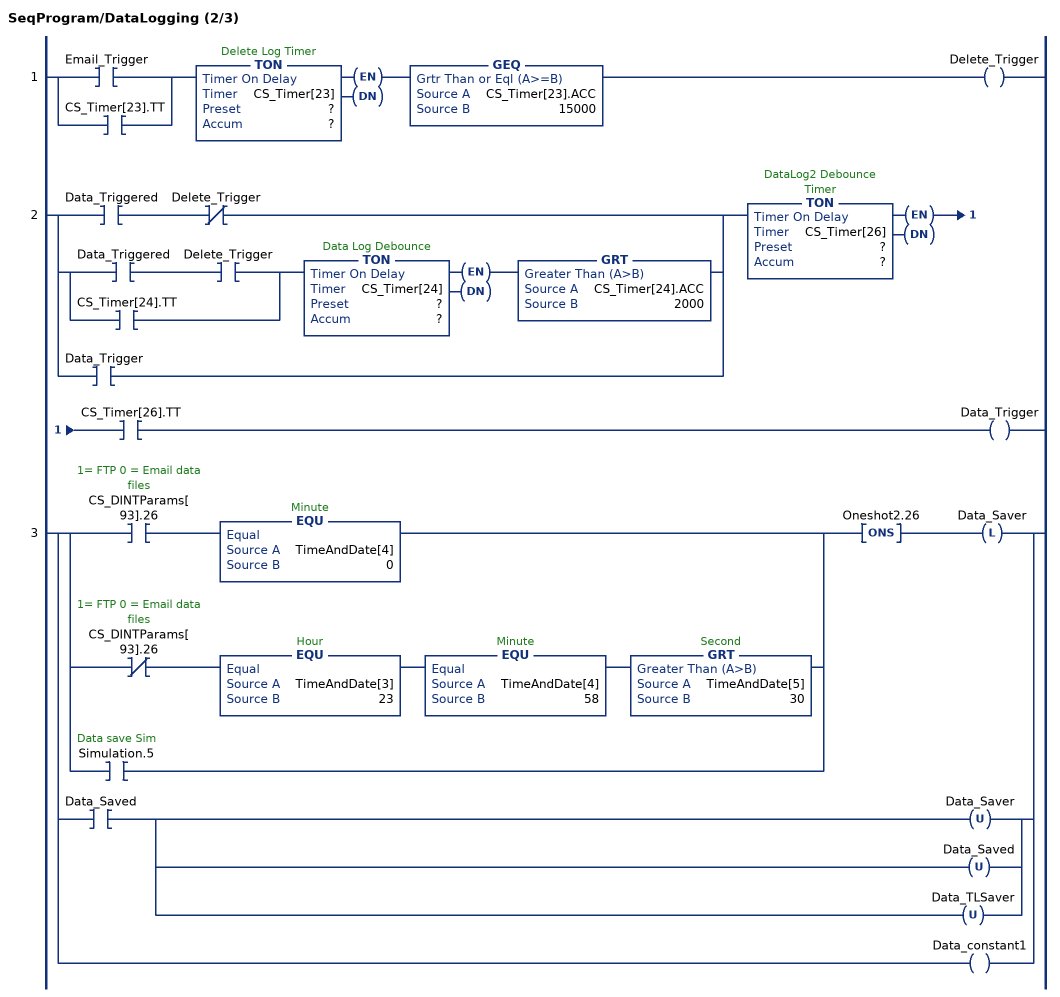
   1: [XIC(Email_Trigger) ,XIC(CS_Timer[23].TT) ]TON(CS_Timer[23],?,?)GEQ(CS_Timer[23].ACC,15000)OTE(Delete_Trigger);
   2: [[XIC(Data_Triggered) XIO(Delete_Trigger) ,[XIC(Data_Triggered) XIC(Delete_Trigger) ,XIC(CS_Timer[24].TT) ] TON(CS_Timer[24],?,?) GRT(CS_Timer[24].ACC,2000) ] ,XIC(Data_Trigger) ]TON(CS_Timer[26],?,?)XIC(CS_Timer[26].TT)OTE(Data_Trigger);
   3: [[XIC(CS_DINTParams[93].26) EQU(TimeAndDate[4],0) ,XIO(CS_DINTParams[93].26) EQU(TimeAndDate[3],23) EQU(TimeAndDate[4],58) GRT(TimeAndDate[5],30) ,XIC(Simulation.5) ] ONS(Oneshot2.26) OTL(Data_Saver) ,XIC(Data_Saved) [OTU(Data_Saver) ,OTU(Data_Saved) ,OTU(Data_TLSaver) ] ,OTE(Data_constant1) ];
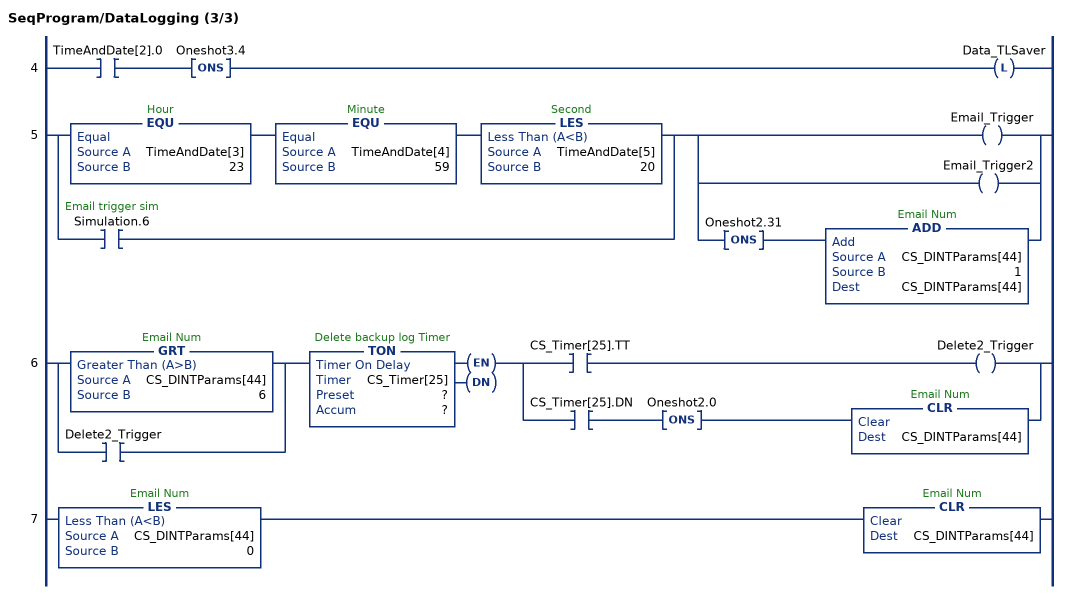
   4: XIC(TimeAndDate[2].0)ONS(Oneshot3.4)OTL(Data_TLSaver);
   5: [EQU(TimeAndDate[3],23) EQU(TimeAndDate[4],59) LES(TimeAndDate[5],20) ,XIC(Simulation.6) ][[OTE(Email_Trigger) ,OTE(Email_Trigger2) ] ,ONS(Oneshot2.31) ADD(CS_DINTParams[44],1,CS_DINTParams[44]) ];
   6: [GRT(CS_DINTParams[44],6) ,XIC(Delete2_Trigger) ]TON(CS_Timer[25],?,?)[XIC(CS_Timer[25].TT) OTE(Delete2_Trigger) ,XIC(CS_Timer[25].DN) ONS(Oneshot2.0) CLR(CS_DINTParams[44]) ];
   7: LES(CS_DINTParams[44],0)CLR(CS_DINTParams[44]);
END_ROUTINE
